{attribute 'qualified_only'}
VAR_GLOBAL

	stTrafficInArray : ARRAY[1..4] OF ST_TrafficLightInput;
	stTrafficOutArray : ARRAY[1..4] OF ST_TrafficLightOutput;

END_VAR

(* stored: Version 1.1.0.1, ProductVersion 3.1.4024.0
   GVL TrafficLightGVL: Id {976dfae4-6008-4f08-9ee3-1f3430a5e16d} *)
